FUNCTION F_TargetReachedOrLower : BOOL
VAR_INPUT
	fCurrentPos: LREAL;
	fTargetPos: LREAL;
END_VAR


F_TargetReachedOrLower := fCurrentPos <= (fTargetPos + fEpsilon);

END_FUNCTION

(* stored: Version 1.1.0.1, ProductVersion 3.1.4020.12
   POU F_TargetReachedOrLower: Id {4cd65146-0c1a-48df-a4a3-8832351a5c41}, SpecialFunc None *)
